INTERFACE I_Cylinder

METHOD Extend
VAR_INPUT
END_VAR
END_METHOD

PROPERTY Extended : BOOL
GET
END_GET
END_PROPERTY

PROPERTY ExtendTime : LREAL
GET
END_GET
SET
END_SET
END_PROPERTY

METHOD Retract
VAR_INPUT
END_VAR
END_METHOD

PROPERTY Retracted : BOOL
GET
END_GET
END_PROPERTY

PROPERTY RetractTime : LREAL
GET
END_GET
SET
END_SET
END_PROPERTY

END_INTERFACE

(* stored: Version 1.1.0.1
   Itf I_Cylinder: Id {50ca6ff3-f8de-4812-b33f-a125edbe41cc}
   Method Extend: Id {6fbcc9e0-be52-4e2a-9078-3acec51c193a}
   Property Extended: Id {9f4d9bef-6c2c-4f9e-ab74-6501c7dcdd54}
   Get Get: Id {0ce0f491-727f-46bd-8ae9-d07fc1b439f4}
   Property ExtendTime: Id {0b25d1f7-7d2b-4293-927e-c976acf84c90}
   Get Get: Id {a9d984a8-e2c9-4448-8b87-030a9d7ace95}
   Set Set: Id {b8aa82ed-a8e6-4c73-86f0-2dea90f4093e}
   Method Retract: Id {e9f314be-8bc7-45b6-badc-a8667edfcee4}
   Property Retracted: Id {d3c1ed2b-0f2f-45fa-8b47-63220b6c1c72}
   Get Get: Id {432d6e09-2b85-489a-899f-8c5f849d134c}
   Property RetractTime: Id {39f45264-4659-40f9-aa89-df4bfa2eedd2}
   Get Get: Id {a3fd9ea1-b55a-4ccd-9c5b-728a04948787}
   Set Set: Id {3fc0243a-2e25-4d04-a19a-68b7bec5a887} *)
